PROGRAM MAIN
VAR
END_VAR

END_PROGRAM

(* stored: Version 1.1.0.1, ProductVersion 3.1.0.36
   POU MAIN: Id {273e6257-77ca-40bb-8b4b-eee03fb49dd5}, SpecialFunc None *)
